FUNCTION_BLOCK Starting_State  IMPLEMENTS ITF_State
VAR_INPUT
END_VAR
VAR_OUTPUT
END_VAR
VAR
	pPML_Base : POINTER TO PML_StatePattern_Base;
	_stateMachine : IPmlStateMachine;
END_VAR

METHOD Cycle : BOOL
VAR_INPUT
END_VAR
_stateMachine.SetStateComplete();
pPML_Base^.SetState(pPML_Base^.execute);
END_METHOD

METHOD FB_init : BOOL
VAR_INPUT
	bInitRetains : BOOL; // if TRUE, the retain variables are initialized (warm start / cold start)
	bInCopyCode : BOOL;  // if TRUE, the instance afterwards gets moved into the copy code (online change)
	pPML_Base : POINTER TO PML_StatePattern_Base;
	statemachine : IPmlStateMachine;
END_VAR
_stateMachine := statemachine;
THIS^.pPML_Base := pPML_Base;
END_METHOD

END_FUNCTION_BLOCK

(* stored: Version 1.1.0.1, ProductVersion 3.1.4024.12
   POU Starting_State: Id {254cf892-dba0-45be-b7ba-aaead1a53f14}, SpecialFunc None
   Method Cycle: Id {4cf13cf2-2104-4b83-90d0-2da1c4090901}
   Method FB_init: Id {0c0aa8b5-6c94-493c-b0a4-4654db3bcb60} *)
